{attribute 'qualified_only'}
VAR_GLOBAL
	Axis: AXIS_REF;
	pAbilitaMotore: BOOL;
	pDisabilitaMotore: BOOL;
	motoreAbilitato: BOOL;
	pAbilitaJog: BOOL;
	bErrorJog: BOOL;
	pMoveVelocity: BOOL;
	pHalt: BOOL;
END_VAR

(* stored: Version 1.1.0.1, ProductVersion 3.1.4024.12
   GVL GVL: Id {75970409-6cef-43b3-8ebe-a18c6cf1903e} *)
